// TIA Portal V16 export
// export: Created 2024-09-05T17:39:05.449257Z, ExportSetting WithDefaults, DisplayName Totally Integrated Automation Portal, DisplayVersion V16 Update 6, DisplayName TIA Portal Version Control Interface, DisplayVersion V16 Update 2, DisplayName TIA Portal Openness, DisplayVersion V16 Update 6, DisplayName STEP 7 Professional, DisplayVersion V16 Update 6, DisplayName STEP 7 Safety, DisplayVersion V16, DisplayName WinCC Advanced, DisplayVersion V16 Update 6
FUNCTION_BLOCK "CylinderINC"   // FB30, LAD
{ S7_Optimized_Access := 'FALSE' }
AUTHOR : Bodorik
FAMILY : RIV
NAME : Cylinder
VERSION : 0.9
// stored: AutoNumber false, IsIECCheckEnabled false, SetENOAutomatically false, UDAEnableTagReadback false
   VAR_INPUT
      POWER_OK : Bool;
      MOVE_BASIC : Bool;
      MOVE_WORK : Bool;
      MOVE_FREE : Bool;   // QB 5
      BASIC_POSITION : Bool;   // Save cycle time
      WORK_POSITION : Bool;
      TRIGGER : Bool;
      RESET : Bool;   // QB 3
      DELAY_BASIC : Time := T#1S;
      DELAY_WORK : Time := T#1S;
      DELAY_FREE : Time := T#1S;
      ERROR_TIME : Time := T#1S;
      ValveDelay : Time;
   END_VAR
   VAR_OUTPUT
      VALVE_BASIC : Bool;   // Taking nut
      VALVE_WORK : Bool;   // 'Operate' authorization.
      CylinderStatus : "CylinderStatus";
      ERROR_BASIC : Bool;
      ERROR_WORK : Bool;
   END_VAR
   VAR_IN_OUT
      CylinderOperation : "CylinderOperation";
   END_VAR
   VAR DB_SPECIFIC
      "4l+Started" : Bool;
      InitCommandBP : Bool;
      InitCommandWP : Bool;
      BasicWorkStartWP : Bool;
      BasicWorkStartBP : Bool;
      work_valve : Bool;
      basic_valve : Bool;   // In working position
      free_valve : Bool;
      baspos_error { S7_SetPoint := 'True'} : TON_TIME;   // ton db
      workpos_error { S7_SetPoint := 'True'} : TON_TIME;
      baspos_delay { S7_SetPoint := 'True'} : TON_TIME;
      workpos_delay { S7_SetPoint := 'True'} : TON_TIME;
      CylinderOperationOld { S7_SetPoint := 'True'} : "CylinderOperation";
      IEC_Timer_0_Instance { S7_SetPoint := 'True'} : TP_TIME;
   END_VAR
   VAR
      R_TRIG_Instance { S7_SetPoint := 'True'} : R_TRIG;
   END_VAR
   VAR DB_SPECIFIC
      IEC_Timer_0_Instance_1 { S7_SetPoint := 'True'} : TP_TIME;
      IEC_Timer_0_Instance_2 { S7_SetPoint := 'True'} : TP_TIME;
      IEC_Timer_0_Instance_3 { S7_SetPoint := 'True'} : TON_TIME;
      IEC_Timer_0_Instance_4 { S7_SetPoint := 'True'} : TON_TIME;
   END_VAR
   VAR_TEMP
      et : Bool;
   END_VAR
   VAR_TEMP   // added for the SCL form of the ladder/FBD networks
      _w1 : Bool;
   END_VAR
BEGIN

REGION Network 1 (SCL): check new cylinder command
   //check if basic position req movement changed
   IF #CylinderOperation.ToBp <> #CylinderOperationOld.ToBp THEN
       #CylinderOperation.ToFp := false;
       #CylinderOperation.ToWp := false;
   END_IF;
   //check if work position req movement changed
   IF #CylinderOperation.ToWp <> #CylinderOperationOld.ToWp THEN
       #CylinderOperation.ToFp := false;
       #CylinderOperation.ToBp := false;
   END_IF;
   //check if free position req movement changed
   IF #CylinderOperation.ToFp <> #CylinderOperationOld.ToFp THEN
       #CylinderOperation.ToBp := false;
       #CylinderOperation.ToWp := false;
   END_IF;
   //store actual cylinder status to old
   #CylinderOperationOld := #CylinderOperation;
END_REGION

REGION Network 2: Start movement to basic position
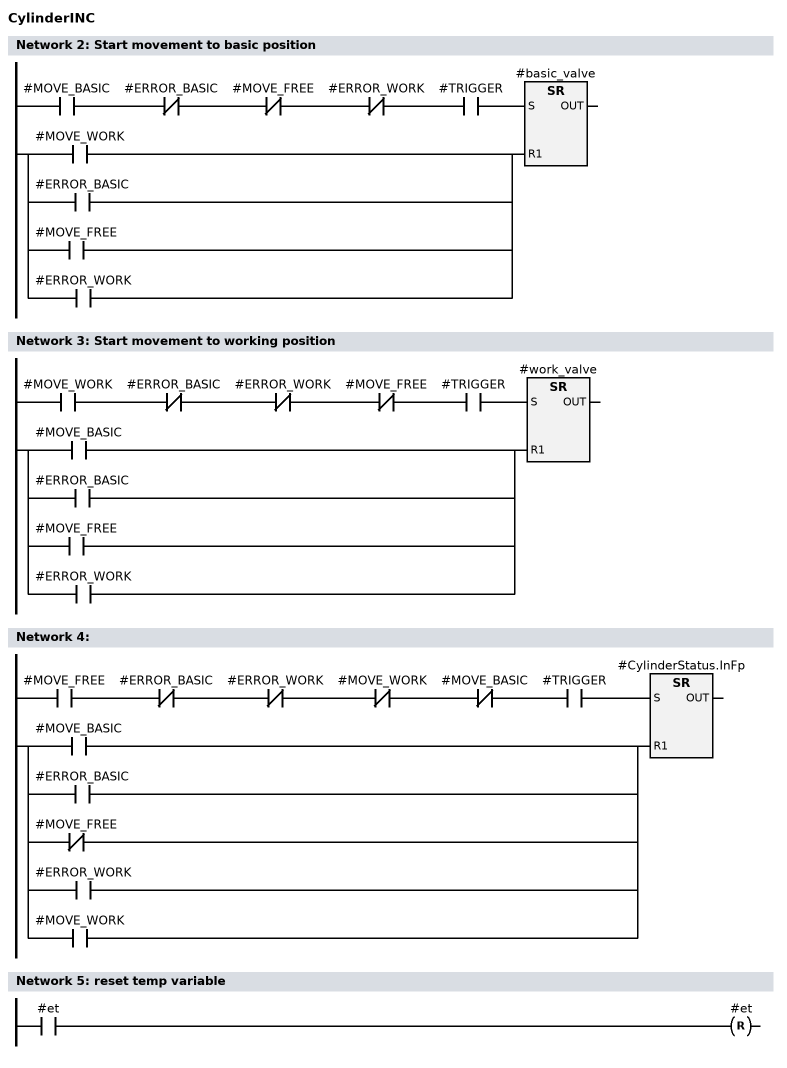
   RUNG wire#powerrail
      Contact( #MOVE_BASIC )
      I_Contact( #ERROR_BASIC )
      I_Contact( #MOVE_FREE )
      I_Contact( #ERROR_WORK )
      Contact( #TRIGGER )
      S_SR(operand := #basic_valve, r1 := wire#w1)
   END_RUNG
   RUNG wire#powerrail
      Contact( #MOVE_WORK )
   END_RUNG wire#w1
   RUNG wire#powerrail
      Contact( #ERROR_BASIC )
   END_RUNG wire#w1
   RUNG wire#powerrail
      Contact( #MOVE_FREE )
   END_RUNG wire#w1
   RUNG wire#powerrail
      Contact( #ERROR_WORK )
   END_RUNG wire#w1
   // the same network as SCL:
   IF #MOVE_BASIC AND NOT #ERROR_BASIC AND NOT #MOVE_FREE AND NOT #ERROR_WORK AND #TRIGGER THEN
       #basic_valve := TRUE;   // SR flip-flop
   END_IF;
   IF #MOVE_WORK OR #ERROR_BASIC OR #MOVE_FREE OR #ERROR_WORK THEN #basic_valve := FALSE; END_IF;
END_REGION

REGION Network 3: Start movement to working position
   RUNG wire#powerrail
      Contact( #MOVE_WORK )
      I_Contact( #ERROR_BASIC )
      I_Contact( #ERROR_WORK )
      I_Contact( #MOVE_FREE )
      Contact( #TRIGGER )
      S_SR(operand := #work_valve, r1 := wire#w1)
   END_RUNG
   RUNG wire#powerrail
      Contact( #MOVE_BASIC )
   END_RUNG wire#w1
   RUNG wire#powerrail
      Contact( #ERROR_BASIC )
   END_RUNG wire#w1
   RUNG wire#powerrail
      Contact( #MOVE_FREE )
   END_RUNG wire#w1
   RUNG wire#powerrail
      Contact( #ERROR_WORK )
   END_RUNG wire#w1
   // the same network as SCL:
   IF #MOVE_WORK AND NOT #ERROR_BASIC AND NOT #ERROR_WORK AND NOT #MOVE_FREE AND #TRIGGER THEN
       #work_valve := TRUE;   // SR flip-flop
   END_IF;
   IF #MOVE_BASIC OR #ERROR_BASIC OR #MOVE_FREE OR #ERROR_WORK THEN #work_valve := FALSE; END_IF;
END_REGION

REGION Network 4
   RUNG wire#powerrail
      Contact( #MOVE_FREE )
      I_Contact( #ERROR_BASIC )
      I_Contact( #ERROR_WORK )
      I_Contact( #MOVE_WORK )
      I_Contact( #MOVE_BASIC )
      Contact( #TRIGGER )
      S_SR(operand := #CylinderStatus.InFp, r1 := wire#w1)
   END_RUNG
   RUNG wire#powerrail
      Contact( #MOVE_BASIC )
   END_RUNG wire#w1
   RUNG wire#powerrail
      Contact( #ERROR_BASIC )
   END_RUNG wire#w1
   RUNG wire#powerrail
      I_Contact( #MOVE_FREE )
   END_RUNG wire#w1
   RUNG wire#powerrail
      Contact( #ERROR_WORK )
   END_RUNG wire#w1
   RUNG wire#powerrail
      Contact( #MOVE_WORK )
   END_RUNG wire#w1
   // the same network as SCL:
   IF #MOVE_FREE AND NOT #ERROR_BASIC AND NOT #ERROR_WORK AND NOT #MOVE_WORK AND NOT #MOVE_BASIC AND #TRIGGER THEN
       #CylinderStatus.InFp := TRUE;   // SR flip-flop
   END_IF;
   IF #MOVE_BASIC OR #ERROR_BASIC OR NOT #MOVE_FREE OR #ERROR_WORK OR #MOVE_WORK THEN
       #CylinderStatus.InFp := FALSE;
   END_IF;
END_REGION

REGION Network 5: reset temp variable
   RUNG wire#powerrail
      Contact( #et )
      R_Coil( #et )
   END_RUNG
   // the same network as SCL:
   IF #et THEN #et := FALSE; END_IF;
END_REGION

REGION Network 6 (FBD): Error movement to basic position
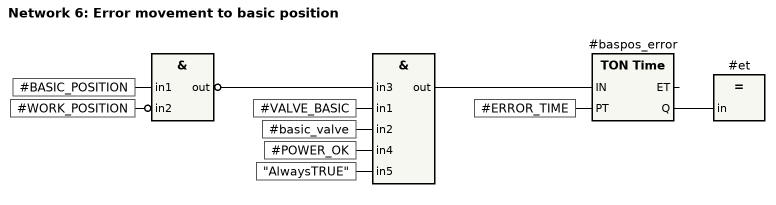
   #baspos_error(IN := NOT (#BASIC_POSITION AND NOT #WORK_POSITION) AND #VALVE_BASIC AND #basic_valve AND #POWER_OK AND "AlwaysTRUE",   // TON
                 PT := #ERROR_TIME);
   #et := #baspos_error.Q;
END_REGION

REGION Network 7: Set basic position error
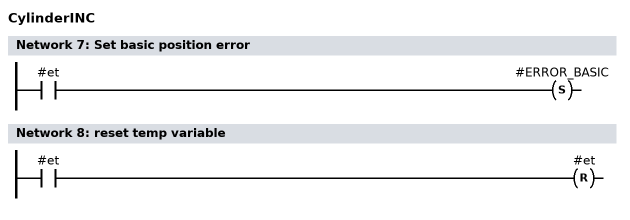
   RUNG wire#powerrail
      Contact( #et )
      S_Coil( #ERROR_BASIC )
   END_RUNG
   // the same network as SCL:
   IF #et THEN #ERROR_BASIC := TRUE; END_IF;
END_REGION

REGION Network 8: reset temp variable
   RUNG wire#powerrail
      Contact( #et )
      R_Coil( #et )
   END_RUNG
   // the same network as SCL:
   IF #et THEN #et := FALSE; END_IF;
END_REGION

REGION Network 9 (FBD): Error movement to working position
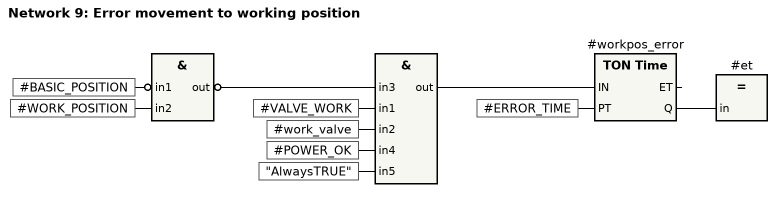
   #workpos_error(IN := NOT (NOT #BASIC_POSITION AND #WORK_POSITION) AND #VALVE_WORK AND #work_valve AND #POWER_OK AND "AlwaysTRUE",   // TON
                  PT := #ERROR_TIME);
   #et := #workpos_error.Q;
END_REGION

REGION Network 10: Set working position error
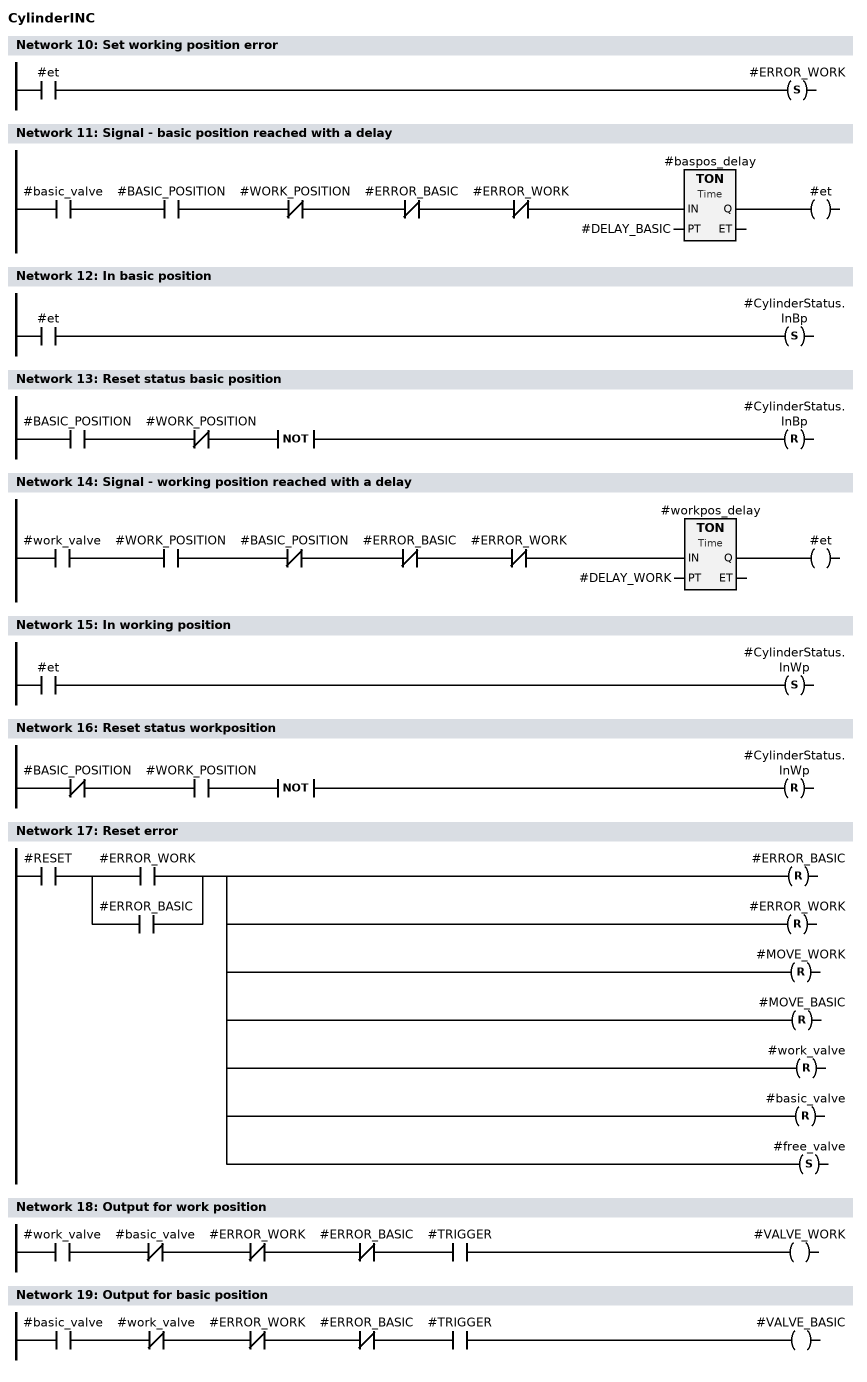
   RUNG wire#powerrail
      Contact( #et )
      S_Coil( #ERROR_WORK )
   END_RUNG
   // the same network as SCL:
   IF #et THEN #ERROR_WORK := TRUE; END_IF;
END_REGION

REGION Network 11: Signal - basic position reached with a delay
   RUNG wire#powerrail
      Contact( #basic_valve )
      Contact( #BASIC_POSITION )
      I_Contact( #WORK_POSITION )
      I_Contact( #ERROR_BASIC )
      I_Contact( #ERROR_WORK )
      { S7_Templates := "time_type := Time" } #baspos_delay.TON(pt := #DELAY_BASIC, et =>)
      Coil( #et )
   END_RUNG
   // the same network as SCL:
   #baspos_delay(PT := #DELAY_BASIC,   // TON
                 IN := #basic_valve AND #BASIC_POSITION AND NOT #WORK_POSITION AND NOT #ERROR_BASIC AND NOT #ERROR_WORK);
   #et := #baspos_delay.Q;
END_REGION

REGION Network 12: In basic position
   RUNG wire#powerrail
      Contact( #et )
      S_Coil( #CylinderStatus.InBp )
   END_RUNG
   // the same network as SCL:
   IF #et THEN #CylinderStatus.InBp := TRUE; END_IF;
END_REGION

REGION Network 13: Reset status basic position
   RUNG wire#powerrail
      Contact( #BASIC_POSITION )
      I_Contact( #WORK_POSITION )
      Not()
      R_Coil( #CylinderStatus.InBp )
   END_RUNG
   // the same network as SCL:
   IF NOT (#BASIC_POSITION AND NOT #WORK_POSITION) THEN #CylinderStatus.InBp := FALSE; END_IF;
END_REGION

REGION Network 14: Signal - working position reached with a delay
   RUNG wire#powerrail
      Contact( #work_valve )
      Contact( #WORK_POSITION )
      I_Contact( #BASIC_POSITION )
      I_Contact( #ERROR_BASIC )
      I_Contact( #ERROR_WORK )
      { S7_Templates := "time_type := Time" } #workpos_delay.TON(pt := #DELAY_WORK, et =>)
      Coil( #et )
   END_RUNG
   // the same network as SCL:
   #workpos_delay(PT := #DELAY_WORK,   // TON
                  IN := #work_valve AND #WORK_POSITION AND NOT #BASIC_POSITION AND NOT #ERROR_BASIC AND NOT #ERROR_WORK);
   #et := #workpos_delay.Q;
END_REGION

REGION Network 15: In working position
   RUNG wire#powerrail
      Contact( #et )
      S_Coil( #CylinderStatus.InWp )
   END_RUNG
   // the same network as SCL:
   IF #et THEN #CylinderStatus.InWp := TRUE; END_IF;
END_REGION

REGION Network 16: Reset status workposition
   RUNG wire#powerrail
      I_Contact( #BASIC_POSITION )
      Contact( #WORK_POSITION )
      Not()
      R_Coil( #CylinderStatus.InWp )
   END_RUNG
   // the same network as SCL:
   IF NOT (NOT #BASIC_POSITION AND #WORK_POSITION) THEN #CylinderStatus.InWp := FALSE; END_IF;
END_REGION

REGION Network 17: Reset error
   RUNG wire#powerrail
      Contact( #RESET )
      wire#w1
      Contact( #ERROR_WORK )
      wire#w2
      R_Coil( #ERROR_BASIC )
   END_RUNG
   RUNG wire#w1
      Contact( #ERROR_BASIC )
   END_RUNG wire#w2
   RUNG wire#w2
      R_Coil( #ERROR_WORK )
   END_RUNG
   RUNG wire#w2
      R_Coil( #MOVE_WORK )
   END_RUNG
   RUNG wire#w2
      R_Coil( #MOVE_BASIC )
   END_RUNG
   RUNG wire#w2
      R_Coil( #work_valve )
   END_RUNG
   RUNG wire#w2
      R_Coil( #basic_valve )
   END_RUNG
   RUNG wire#w2
      S_Coil( #free_valve )
   END_RUNG
   // the same network as SCL:
   #_w1 := #RESET AND (#ERROR_WORK OR #ERROR_BASIC);
   IF #_w1 THEN
       #ERROR_BASIC := FALSE;
       #ERROR_WORK := FALSE;
       #MOVE_WORK := FALSE;
       #MOVE_BASIC := FALSE;
       #work_valve := FALSE;
       #basic_valve := FALSE;
       #free_valve := TRUE;
   END_IF;
END_REGION

REGION Network 18: Output for work position
   RUNG wire#powerrail
      Contact( #work_valve )
      I_Contact( #basic_valve )
      I_Contact( #ERROR_WORK )
      I_Contact( #ERROR_BASIC )
      Contact( #TRIGGER )
      Coil( #VALVE_WORK )
   END_RUNG
   // the same network as SCL:
   #VALVE_WORK := #work_valve AND NOT #basic_valve AND NOT #ERROR_WORK AND NOT #ERROR_BASIC AND #TRIGGER;
END_REGION

REGION Network 19: Output for basic position
   RUNG wire#powerrail
      Contact( #basic_valve )
      I_Contact( #work_valve )
      I_Contact( #ERROR_WORK )
      I_Contact( #ERROR_BASIC )
      Contact( #TRIGGER )
      Coil( #VALVE_BASIC )
   END_RUNG
   // the same network as SCL:
   #VALVE_BASIC := #basic_valve AND NOT #work_valve AND NOT #ERROR_WORK AND NOT #ERROR_BASIC AND #TRIGGER;
END_REGION

REGION Network 20 (SCL)
   #R_TRIG_Instance(CLK:=#POWER_OK
   );

   IF #R_TRIG_Instance.Q THEN
       #"4l+Started" := TRUE;

   END_IF;

   IF #MOVE_BASIC AND #"4l+Started" THEN

       #InitCommandBP := true;
   END_IF;
   IF #MOVE_WORK AND #"4l+Started" THEN

       #InitCommandWP := true;
   END_IF;

   #IEC_Timer_0_Instance_1(IN:=#InitCommandBP,
                               PT:=t#10ms,
                               Q=>#BasicWorkStartBP
       );
   #IEC_Timer_0_Instance_2(IN:=#InitCommandWP,
                               PT:=t#10ms,
                               Q=>#BasicWorkStartWP
   );


   IF #BasicWorkStartBP  THEN
       #VALVE_WORK := TRUE;
       #VALVE_BASIC := FALSE;
       ;

   END_IF;

   IF #BasicWorkStartWP THEN
       #VALVE_WORK := FALSE;
       #VALVE_BASIC := TRUE;
       ;

   END_IF;

   IF NOT #IEC_Timer_0_Instance_1.Q AND #InitCommandBP THEN
       #VALVE_WORK := FALSE;
       #VALVE_BASIC := TRUE;
       #"4l+Started" := FALSE;
       #InitCommandBP := FALSE;
       ;
   END_IF;
   IF NOT #IEC_Timer_0_Instance_2.Q AND #InitCommandWP THEN
       #VALVE_WORK := TRUE;
       #VALVE_BASIC := FALSE;
       #"4l+Started" := FALSE;
       #InitCommandWP := FALSE;
       ;
   END_IF;
END_REGION
END_FUNCTION_BLOCK
